FUNCTION_BLOCK TcpServer_Test EXTENDS FB_TestSuite
VAR
	startTcpServerTest		: BOOL;
	tcpServerTestDone		: BOOL;
	tcpServerTestTimeout	: TON := (PT:= T#2M);
	
	tcpServer	: TcTcpServer(BufferSize:= TcTcpUdpRT_Param.RingBufferSize);
	listenPort	: UINT := 9900;
	txData		: STRING(25) := 'Hello from PLC TCP server';
	txCounter	: UDINT;
	rxData		: STRING;
	rxCounter	: UDINT;
	methodTimeout		: TON;
END_VAR

tcpServer.Run();

IF startTcpServerTest THEN
	OpenConnectionAndListenForClient();
	WaitForTcpClientToConnect();
	ReceiveDataFromTcpClient();
	SendDataToTcpClient();
	WaitForClientToDisconnect();
END_IF

TEST('RunTcpServerTest');
tcpServerTestTimeout(IN:= startTcpServerTest);
IF tcpServerTestDone THEN
	tcpServerTestTimeout(IN:= FALSE);
	TEST_FINISHED();
ELSIF tcpServerTestTimeout.Q THEN
	AssertFalse(Condition:= tcpServerTestTimeout.Q, Message:= 'TcpServer_Test timed out while running');
	tcpServerTestTimeout(IN:= FALSE);
	TEST_FINISHED();
ELSIF tcpServer.Error THEN
	AssertFalse(Condition:= tcpServer.Error, Message:= tcpServer.GetError);
	tcpServerTestTimeout(IN:= FALSE);
	TEST_FINISHED();
END_IF

METHOD OpenConnectionAndListenForClient
VAR_INST
	openConnection: BOOL;
END_VAR
IF TEST_ORDERED('OpenConnectionAndListenForClient') THEN
	openConnection := tcpServer.OpenConnection(listenPort);
	AssertTrue(Condition:= openConnection, Message:= 'Failed to open TCP server connection');
	TEST_FINISHED();	
END_IF
END_METHOD

METHOD ReceiveDataFromTcpClient
VAR_INST
	delay: TIME := T#15S;
END_VAR
IF TEST_ORDERED('ReceiveDataFromTcpClient') THEN
	methodTimeout(IN:= TRUE, PT:= delay);
	IF tcpServer.IsDataAvailable THEN
		IF tcpServer.Receive(DataPointer:= ADR(rxData), DataLength:= SIZEOF(rxData), ReceivedLength=> rxCounter) THEN
			ADSLOGSTR(msgCtrlMask:= ADSLOG_MSGTYPE_LOG, msgFmtStr:= 'Message received: %s', strArg:= rxData);
			AssertTrue(Condition:= rxCounter > 0, Message:= 'The data from the TCP client had a length of zero');
			methodTimeout(IN:= FALSE);
			TEST_FINISHED();
		END_IF
	ELSIF methodTimeout.Q THEN
		AssertTrue(Condition:= FALSE, Message:= 'TCP server timed out waiting for data from the TCP client');
		methodTimeout(IN:= FALSE);
		TEST_FINISHED();
	END_IF
END_IF
END_METHOD

METHOD SendDataToTcpClient
VAR_INST
	delay: TIME := T#15S;
END_VAR
IF TEST_ORDERED('SendDataToTcpClient') THEN
	methodTimeout(IN:= TRUE, PT:= delay);
	IF tcpServer.Send(DataPointer:= ADR(txData), DataLength:= SIZEOF(txData), DataSent=> txCounter) THEN
		ADSLOGSTR(msgCtrlMask:= ADSLOG_MSGTYPE_LOG, msgFmtStr:= 'Message sent: %s', strArg:= txData);
		AssertTrue(Condition:= txCounter > 0, Message:= 'The data sent to the TCP client had a length of zero');
		methodTimeout(IN:= FALSE);
		TEST_FINISHED();
	ELSIF methodTimeout.Q THEN
		AssertTrue(Condition:= FALSE, Message:= 'TCP server timed out sending data to the TCP client');
		methodTimeout(IN:= FALSE);
		TEST_FINISHED();
	END_IF
END_IF
END_METHOD

METHOD WaitForClientToDisconnect
VAR_INST
	delay: TIME := T#15S;
END_VAR
IF TEST_ORDERED('WaitForClientToDisconnect') THEN
	methodTimeout(IN:= TRUE, PT:= delay);
	IF NOT  tcpServer.IsConnected THEN
		tcpServerTestDone := TRUE;
		methodTimeout(IN:= FALSE);
		TEST_FINISHED();
	ELSIF methodTimeout.Q THEN
		AssertTrue(Condition:= FALSE, Message:= 'TCP server timed out waiting for TCP client to disconnection');
		methodTimeout(IN:= FALSE);
		TEST_FINISHED();
	END_IF
END_IF
END_METHOD

METHOD WaitForTcpClientToConnect
VAR_INST
	delay: TIME := T#15S;
END_VAR
IF TEST_ORDERED('WaitForTcpClientToConnect') THEN
	methodTimeout(IN:= TRUE, PT:= delay);
	IF tcpServer.IsConnected THEN
		methodTimeout(IN:= FALSE);
		TEST_FINISHED();
	ELSIF methodTimeout.Q THEN
		AssertTrue(Condition:= FALSE, Message:= 'TCP server timed out waiting for the TCP client to connection');
		methodTimeout(IN:= FALSE);
		TEST_FINISHED();
	END_IF
END_IF
END_METHOD

END_FUNCTION_BLOCK

(* stored: Version 1.1.0.1
   POU TcpServer_Test: Id {7356ce97-5fa9-0d40-182f-40a6d651e3e8}, SpecialFunc None
   Method OpenConnectionAndListenForClient: Id {42e72aa7-fbb5-075d-08b7-6dad45207f77}
   Method ReceiveDataFromTcpClient: Id {e17060f2-cdc0-06b1-33cb-6c616973211c}
   Method SendDataToTcpClient: Id {2b7b7141-1bcc-0e99-0403-54f875bd5a33}
   Method WaitForClientToDisconnect: Id {6d403a52-4b69-0b9f-1532-6dd26536a0b1}
   Method WaitForTcpClientToConnect: Id {f20f572d-153d-0531-23e8-ce4fefe06fef} *)
